TYPE IpAdrUnion :
UNION
	ipadrIPStack : UDINT;
	ipadr : ARRAY[0..3] OF BYTE;
END_UNION
END_TYPE

(* stored: Version 1.1.0.1, ProductVersion 3.1.4019.0
   DUT IpAdrUnion: Id {74f50984-7cee-4d59-acb7-443e0a659645} *)
